TYPE Axis :
STRUCT
	
	X: REAL;
	Y: REAL;
	Z: REAL;
	
END_STRUCT
END_TYPE

(* stored: Version 1.1.0.1, ProductVersion 3.1.4024.4
   DUT Axis: Id {6bb03eca-6fae-499f-b650-6be1076abdaf} *)
